// TIA Portal project "scl_3" (V18)

(* hardware
DEVICE "S7-1200 station_1"  S7-1200 Station
   slot 0: "Rack_0"  S7-1200 Rack  Rack  V1.0
   slot 1: "PLC_1"  CPU 1214C DC/DC/DC  6ES7 214-1AG40-0XB0  V4.6
*)

// ===== PLC "PLC_1"  CPU 1214C DC/DC/DC =====

VAR_GLOBAL   // PLC tag table "Default tag table"
   "POMPA MOTORU" AT %Q0.0 : Bool;
   "SENSÖR" AT %IW64 : Word;
END_VAR

FUNCTION "Block_1" : Void   // FC1, SCL
{ S7_Optimized_Access := 'TRUE' }
VERSION : 0.1
BEGIN
   "POMPA MOTORU" := ("SENSÖR" > 4500) AND ("SENSÖR" < 20000);
END_FUNCTION

ORGANIZATION_BLOCK "Main"   // OB1, LAD, ProgramCycle
TITLE = "Main Program Sweep (Cycle)"
{ S7_Optimized_Access := 'TRUE' }
VERSION : 0.1
// UGULAMA-2: Bir tanktaki sivinin alt ve üst seviyeleri belirlenen seviyede ise bir
// pompa motoru çalissin. Limit disinda ise çalismasin. Bu ugulama için bir ultrasonik
// sensör kullanarak analog islem yapilmalidir.
// -*Ultrasonik sensör tank bos iken 0 degerini, tank tam dolu iken 27648 sayisal
// degerini vermektedir.
// - *Sensör gerilim sensörü ise 0...10V, akim sensörü ise 0...20 mA veya 4...20mA verir.
// 10V sayisal karsiligi 27648 veya 20 mA sayisal karsiligi 27648'dir.
   VAR_INPUT
      Initial_Call : Bool;   // Initial call of this OB
      Remanence : Bool;   // =True, if remanent data are available
   END_VAR
BEGIN
END_ORGANIZATION_BLOCK